// TIA Portal V19 export
VAR_GLOBAL   // PLC tag table "D25"
   D25_Lp_EntryReq_LB325 AT %Q300.6 : Bool;   // 274SH1
   D25_Lp_SafetyReset_LB325 AT %Q300.7 : Bool;   // 274SH2
   D25_Pb_EntryReq_LB325 AT %I301.1 : Bool;   // 274SH1
   D25_Pb_SafetyReset_LB325 AT %I301.2 : Bool;   // 274SH2
   D25_Comando_Elettroserratura AT %Q300.4 : Bool;   // 274A1
   D25_Funzione_AUX_Elettroserratura AT %Q300.5 : Bool;   // 274A1
   D25_Cancello_Chiuso AT %I300.7 : Bool;   // 274A1
   D25_Cancello_Bloccato AT %I301.0 : Bool;   // 274A1
   D25_Ls_Os1 AT %I1407.0 : Bool;   // 301DI0 - 274A1
   D25_Ls_Os2 AT %I1407.4 : Bool;   // 301DI4 - 274A1
END_VAR
